FUNCTION_BLOCK FB_UINT_INT (* UINT to INT conversion with limiting *)
  (* Standard: 61499-1-D.1; Classification: Type conversion functions *)
  (* Version 0.1, 2001-08-06, JHC, Rockwell Automation, XML version *)
  (* Version 0.0, 2000-05-01, JHC, Rockwell Automation, SRC version *)
  (* Compiler header: package fb.rt.math; *)
  (* Compiler classdef: class FB_UINT_INT extends FBFunction1 *)
  (* Compiler Java IBM VisualAge 3.0 *)
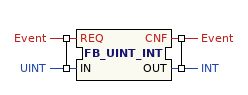
  EVENT_INPUT
    REQ WITH IN;
  END_EVENT
  EVENT_OUTPUT
    CNF WITH OUT;
  END_EVENT
  VAR_INPUT
    IN : UINT;
  END_VAR
  VAR_OUTPUT
    OUT : INT; (* Converted value,-1<OUT<32767 *)
  END_VAR
END_FUNCTION_BLOCK
